Staubli VAL3: Deb2304.pjx

--- Deb2304.pjx ---
Parameters version=s7.4 stackSize=5000 millimeterUnit=true
Program file=Deb2304.pgx
Program file=main.pgx
Program file=start.pgx
Program file=stop.pgx
Data file=Deb2304.dtx

--- main.pgx ---
program main()
begin
  while true
    doECAT1_0 = true

    if(diECAT1_0 == true)

      doECAT1_0 = false

      x[0] = diECAT1_1
      x[1] = diECAT1_2
      x[2] = diECAT1_3
      x[3] = diECAT1_4
      x[4] = diECAT1_5
      x[5] = diECAT1_6
      x[6] = diECAT1_7
      x[7] = diECAT1_8



      y[0] = diECAT1_9
      y[1] = diECAT1_10
      y[2] = diECAT1_11
      y[3] = diECAT1_12
      y[4] = diECAT1_13
      y[5] = diECAT1_14
      y[6] = diECAT1_15
      y[7] = diECAT1_16




      doECAT1_0 = true

    endIf
  endWhile
end
